XA06: CLR   ;
      =     #s_TRS7_Activate; //Then reset the Activate TRS7
      =     #s_TRS8_Activate; //Then reset the Activate TRS8
      =     #o_TRS7_CMD_Req_Run; //Then reset the Run output TRS7
      =     #o_TRS8_CMD_Req_Run; //Then reset the Run output TRS8
      JU    XA99;

XA07: CLR   ;
      =     #s_TRS8_Activate; //Then reset the Activate TRS8
      =     #o_TRS8_CMD_Req_Run; //Then reset the Run output TRS8
      JU    XA99;

XA99: NOP   0;
NETWORK
TITLE =YA: Reporting status to the HLC
//Status is reported on Priority basis:-
//Priority-1. Out of service
//Priority-2. Safety Stop
//Priority-3. Lane is Full (Temporary not available)
//Priority-4. Emptying (Flushing)
//Priority-5. Operational ok & Ready to store the bags on the lane.
//
//If Configured report time(i_CFG_HLC_Report_Time) is more than "0" then status is
//
//reported on configured time interval.
//If Configured report time(i_CFG_HLC_Report_Time) is "0" then status is reported
//on status change.
      L     #i_CFG_HLC_Report_Time; // Load the HLC report time
      L     0;
      ==I   ;
      JCN   YA01;
      R     #s_HLC_Report_Time_Active;
      JU    YA05;

YA01: AN    #s_HLC_Report_Time_Active;
      A(    ;
      L     #s_HLC_Report_Time; // transfer to the memory
      L     0;
      ==I   ;
      )     ;
      JCN   YA02;

      L     #i_CFG_HLC_Report_Time; // Load the HLC report time
      T     #s_HLC_Report_Time; // transfer to the memory

YA02: A     "M_OS_/1.0_sec.";
      JCN   YA05;
      L     #s_HLC_Report_Time;
      L     1;
      -I    ; // THEN delay counter := delay counter
      JPZ   YA03;

// If below zero, then set back at zero
      L     0;
YA03: T     #s_HLC_Report_Time;

      L     #s_HLC_Report_Time; // If the delay time is zero
      L     0;
      <=I   ;
      JCN   YA04; //If it more than zero than jump to the label

      SET   ; // Then cascade delay is done ready to run the motor
      =     #s_HLC_Report_Time_Active;
      JU    YA05;

YA04: CLR   ;
      =     #s_HLC_Report_Time_Active;

//-- Priority -1
YA05: A(    ;
      AN    #o_ST_Operational_On; //Reporting on Time base
      )     ;
      A     #i_Safety_OK;
      A     #s_HLC_Report_Time_Active;
      O(    ;
      A     #o_ST_Operational_On; //Reporting on Status change
      FN    #s_FN_Operation_On;
      A     #i_Safety_OK;
      )     ;
      JCN   YA21;
      L     4; //Reporting "OUT OF SERVICE"
      T     #t_EBS_Lane_State;
      JU    YA20;

//-- Priority -2
YA21: AN    #i_Safety_OK;
      JCN   YA11;

      L     4; // Reporting "OUT OF SERVICE"
      T     #t_EBS_Lane_State;
      JU    YA20;

//-- Priority -3
YA11: A     #o_ST_LSZ_Full; //Reporting on Time base
      A     #s_HLC_Report_Time_Active;
      O(    ;
      A     #o_ST_LSZ_Full; //Reporting on Status change
      FP    #s_FP_LSZ_Full;
      )     ;
      JCN   YA12;
      L     3; //Reporting "LSZ FULL" Temporary Not Available
      T     #t_EBS_Lane_State;
      JU    YA20;

//-- Priority -4
YA12: A     #o_ST_LSZ_Emptying; //Reporting on Time base
      A     #s_HLC_Report_Time_Active;
      O(    ;
      A     #o_ST_LSZ_Emptying; //Reporting on Status change
      FP    #s_FP_LSZ_Emptying;
      )     ;
      JCN   YA13;
      L     2; //Reporting "EMPTYING" Flushing
      T     #t_EBS_Lane_State;
      JU    YA20;

//-- Priority -5
YA13: A     #o_ST_Operational_On; //Reporting on Time base
      AN    #o_ST_LSZ_Full;
      AN    #o_ST_LSZ_Emptying;
      A     #s_HLC_Report_Time_Active;
      O(    ;
      A     #o_ST_Operational_On; //Reporting on Status change
      AN    #o_ST_LSZ_Full;
      AN    #o_ST_LSZ_Emptying;
      FP    #s_FP_Operation_On;
      )     ;
      JCN   YA99;
      L     1; //Reporting "OPERATIONAL" Ready to recieve the Bag
      T     #t_EBS_Lane_State;
      JU    YA20;

YA20: A     #s_HLC_Report_Time_Active; //IF HLC time interval expires
      O(    ; //OR
      L     #t_EBS_Lane_State; //Present EBS Lane State
      L     #s_Prev_Segment_State; //Last report EBS Lane State
      <>I   ; //NOT-EQUAL  Report the EBS Lane State to the DB-Event
      )     ;
      JCN   YA99;

//------------HLC REPORTING-------------//
      CALL "FC_Write_Event" (//Report the EBS Lane State to the DB_Event
           i_Message_ID             := 1404,//EBS Lane Status Report
           i_Event_value            := #t_EBS_Lane_State,
           i_DB_Event_Num           := #t_DB_Event_Num,
           o_Return_Value           := #t_Return_Value);

      L     #t_EBS_Lane_State;
      T     #s_Prev_Segment_State;

      CLR   ;
      =     #s_HLC_Report_Time_Active;

YA99: NOP   0;
NETWORK
TITLE =ZA:Create Availablity Report

      A     #o_ST_Operational_On;
      FP    #s_FP_Operational_Active;
      =     #t_OS_FP_Oper_Active;

      A     #o_ST_Operational_On;
      FN    #s_FN_Operational_Active;
      =     #t_OS_FN_Oper_Active;

      AN    #s_Time_Elapsed_AvaiRep;
      AN    #t_OS_FP_Oper_Active;
      AN    #t_OS_FN_Oper_Active;
      =     #t_StartTimerModereq;

      CALL "FC_On_Dly_Timer_Sec" (
           i_CMD_Start              := #t_StartTimerModereq,
           i_CFG_Timer_Value        := 30,
           i_Setpoint               := #s_TimeSpoint_AvaiRep,
           o_Setpoint               := #s_TimeSpoint_AvaiRep,
           o_Timer_Elapsed          := #s_Time_Elapsed_AvaiRep);


      A     #t_OS_FP_Oper_Active;
      O     #t_OS_FN_Oper_Active;
      O     #s_Time_Elapsed_AvaiRep;
      JCN   ZA99;

      L     0;
      A     #o_ST_Operational_On;
      JCN   ZA01;
      L     1;
ZA01: T     #t_Available_Value;

      CALL "FC_Write_Event" (//Report the EBS Lane State to the DB_Event
           i_Message_ID             := 1221,//Availabilty Report
           i_Event_value            := #t_Available_Value,
           i_DB_Event_Num           := #t_DB_Event_Num,
           o_Return_Value           := #t_Return_Value);

ZA99: NOP   0;
END_FUNCTION_BLOCK

